RoboDK station: DensoAssemblyInverted.rdk

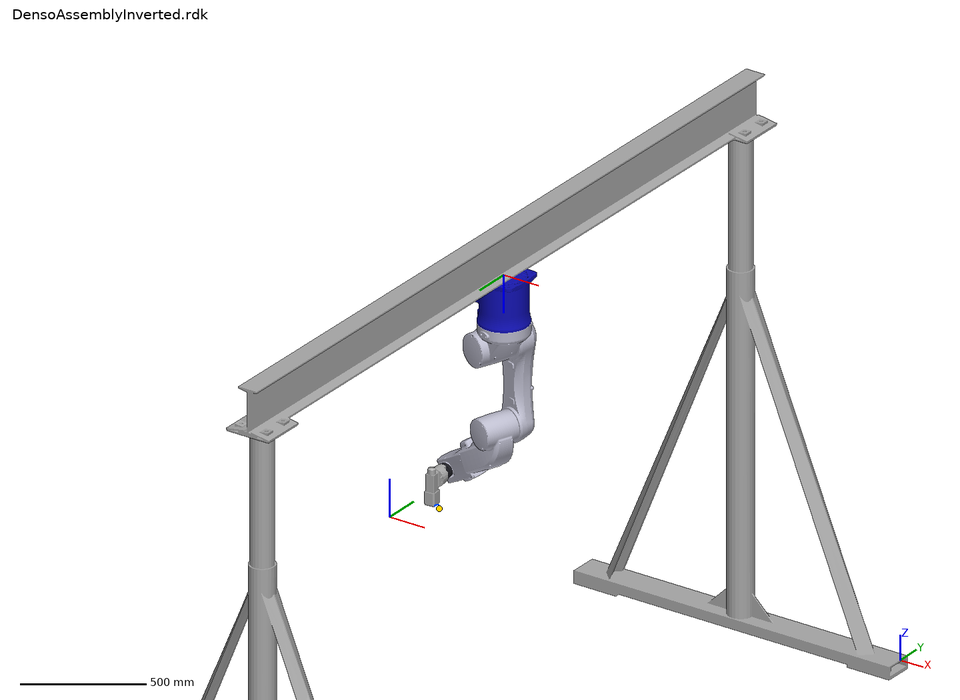
[picture v0: the station drawn from its stored meshes, robots at their saved joint values, targets as dots, program paths as lines]
Station DensoAssemblyInverted (saved by RoboDK 5.5.4). Poses are relative to the parent item; angles as X-Y-Z fixed-axis rotations.
Station parameters (name, value as stored): TAGS, ['Additive Manufacturing', 'Additive manufacturing'], LIN64
  - frame Denso VS-6577G-B Base at (0, 890, 2451.84) mm, rotated rx 180 ry 0 rz 0 deg
    - robot Denso VS-6577G-B: 6 axes, payload 7 kg, reach 854 mm, repeatability 0.03 mm, weight 36 kg
        modified DH rows (alpha deg, a mm, theta deg, d mm): 0, 0, 0, 335; -90, 75, -90, 0; 0, 365, -90, 0; -90, 90, 0, 405; 90, 0, 0, 0; -90, 0, 0, 80
        joint limits [-170, -100, -119, -190, -120, -360] to [170, 135, 169, 190, 120, 360]; home [0, 0, 90, 0, 0, 0]; saved at [-160.107, -3.776, 63.781, -103.06, 111.38, 57.53]
      - tool nozzle, TCP at (110, 10, 80) mm, rotated rx -90 ry 0 rz -90 deg, size 158.8 x 76.2 x 114.9 mm, geometry from nozzle.STEP
  - frame Reference at (-425.65, 710, 1340) mm
    - object Part at (-500, 0, 0) mm, size 120 x 120 x 160 mm, geometry from part.sld
  - machining project Print3D settings: /home/iRETI/RoboticsResearch/WallSection2.gcode | rotZ(0) | rotX(0)*rotY(0) | rotZ(0)
  - Python program Extruder (listed below)
  - Python program SimulateFinalResult (listed below)
  - object Gantry Assembly at (-570, 330, -20) mm, rotated rx 90 ry 0 rz 0 deg, size 1524 x 2402.4 x 3505.2 mm, geometry from Gantry Assembly.STEP
  - program Print3D (214 instructions, listed below)
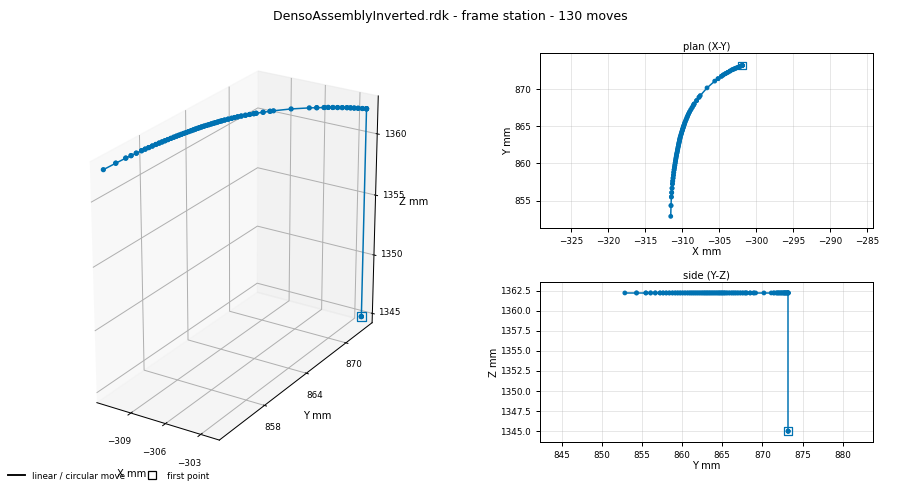
[picture p0: tool path of DensoAssemblyInverted.rdk in frame station, 130 of 130 moves have a stored position in this frame; points joined in program order, loops and branches not executed]

--- Python program Extruder ---
# This macro allows simulating a 3D printing extruder
# The macro will output spray gun statistics
#
# More information about the RoboDK API here:
# https://robodk.com/doc/en/RoboDK-API.html
# For more information visit:
# http://www.robodk.com/doc/en/PythonAPI/robolink.html
#
# Define the default action (0 to deactivate, +1 to activate, -1 to clear any spray gun simulation)
# Setting it to None will display a message
ACTION = None
# Check if we are running this program inside another program and passing arguments
import sys
if len(sys.argv) > 1:
    ACTION = float(sys.argv[1])
    # For faster speed: igone values greater than 0
    if ACTION > 0:
        quit()

from robolink import *    # API to communicate with RoboDK
from robodk import *      # basic matrix operations
RDK = Robolink()

# quit if we are not in simulation mode
if RDK.RunMode() != RUNMODE_SIMULATE:
    quit()

# Get any previously added spray gun simulations and display statistics (spray on the part vs spray falling out of the part)
existing_material_simulation = False
info, stats_data = RDK.Spray_GetStats()
if stats_data.size(1) > 0:
    print("Spray gun statistics:")
    print(info)
    print(stats_data.tr())
    existing_material_simulation = True
    # # Diplay statistics
    # RDK.ShowMessage("Material used: %.1f%%<br>Material waisted: %.1f%%<br>Total particles: %.1f" % (data[1,0],data[2,0],data[3,0]), True)
    # # Clear previous spray
    # RDK.Spray_Clear()

# If the default ACTION is None, display a message to activate/deactivate the spray gun
if ACTION is None:
    print('Note: This macro can be called as Extruder(0) to turn it ON or Extruder(-1) to turn it OFF')
    entry = mbox('Turn Extruder ON or OFF', ('On', '0'), ('Off', '-1'))
    if not entry:
        quit()
    ACTION = int(entry)

if ACTION < 0:
    # Turn material deposition off
    # Select Escape to delete existing material simulations
    #RDK.Spray_Clear()
    RDK.Spray_SetState(SPRAY_OFF)

elif ACTION >= 0:

    if existing_material_simulation:
        # Select Esc key to delete existing material simulations and force a new type of spray gun simulation
        RDK.Spray_SetState(SPRAY_ON)
        exit()


    # Create a new spray gun object in RoboDK for material deposition (3D printing simulation)
    # by using RDK.Spray_Add(tool, object, options_command, volume, geometry)
    # tool: tool item (TCP) to use
    # object: object to project the particles
    # options_command (optional): string to specify options. Example:
    #     STEP=AxB: Defines the grid to be projected 1x1 means only one line of particle projection (for example, for welding)
    #     PARTICLE: Defines the shape and size of particle (sphere or particle), unless a specific geometry is provided:
    #       a- SPHERE(radius, facets)
    #       b- SPHERE(radius, facets, scalex, scaley, scalez)
    #       b- CUBE(sizex, sizey, sizez)
    #     RAND=factor: Defines a random factor factor 0 means that the particles are not deposited randomly
    #     ELLYPSE: defines the volume as an ellypse (default)
    #     RECTANGLE: defines the volume as a rectangle
    #     PROJECT: project the particles to the surface (default) (for welding, painting or scanning)
    #     NO_PROJECT: does not project the particles to the surface (for example, for 3D printing)
    #
    # volume (optional): Matrix of parameters defining the volume of the spray gun
    # geometry (optional): Matrix of vertices defining the triangles.


    diameter = 22.225 # in mm
    detail = 8 # number of rings of detail to display the sphere
    scale = '1,1,0.5' # scale the particle in 0.5 along the tool Z axis (simulating gravity effect)
    options_command = "ELLYPSE NO_PROJECT PARTICLE=SPHERE(%.3f,%.0f,%s)" % (diameter, detail, scale) # simulate
    #options_command = "PARTICLE=CUBE(10,10,2) STEP=8x8"
    #options_command = "PARTICLE=SPHERE(4,8) STEP=8x8"
    #options_command = "PARTICLE=SPHERE(4,8,1,1,0.1) STEP=8x8 RAND=3"

    # Example commands for welding:
    # options_command = "PROJECT PARTICLE=SPHERE(4,8)"
    # options_command = PARTICLE=SPHERE(4,8) STEP=1x0

    tool = 0    # auto detect active tool
    obj = 0     # auto detect object in active reference frame

    # Material is deposited at 0,0,0 with respect to the TCP coordinates
    close_param = [0,0,0,  0,0,0,  0,0,0,     0.7,0.5,0.8,1] # color as RGBA
    far_param   = [0,0,0,  0,0,0,  0,0,0,     0.7,0.5,0.8,1] # color as RGBA
    volume = Mat([close_param, far_param])
    RDK.Spray_Add(tool, obj, options_command, volume.tr())
    RDK.Spray_SetState(SPRAY_ON)

--- Python program SimulateFinalResult ---
# This script will simulate the final result of the 3D printed part using the Spray function

# Or visit: http://www.robodk.com/doc/PythonAPI/
# Note: you do not need to keep a copy of this file, your python script is saved with the station
from robolink import *    # API to communicate with RoboDK
from robodk import *      # basic matrix operations


RENDER = True      # Set to False
STEP_MM = 2         # Detail step in MM for linear moves
STEP_DEG = 2        # Detail step in DEG for joint moves

# Start a connection with the RoboDK API
RDK = Robolink()

# Select the first/only robot in the cell:
program = RDK.ItemUserPick('Select a program to simulate', ITEM_TYPE_PROGRAM)
if not program.Valid():
    raise Exception("No program available")

# Get the robot
robot = RDK.Item('', ITEM_TYPE_ROBOT)
#robot = program.getLink(ITEM_TYPE_ROBOT) # available in newer versions
if not robot.Valid():
    raise Exception("No robot available")

progname = program.Name()
print("Using program %s" % progname)


# Get the program as a list of joint values
tool = robot.getLink(ITEM_TYPE_TOOL)
progok_jlist = program.InstructionListJoints(STEP_MM, STEP_DEG)
progok = progok_jlist[0] # progok: String that indicates if there are any issues with the program
jlist = progok_jlist[1]  # jlist: list of joints

# Check that the program is correct and has at least a movement
njoints = jlist.size(1)
if njoints < 1:
    raise Exception("Program %s has no movements" % name)

# Check if there are any issues with the program:
if progok != "Success":
    raise Exception("Problems with program %s: %s." %(name, progok))

# Reset any material deposition simulation
RDK.Spray_Clear()

robot.setPoseTool(tool)

# Start material deposition simulation according to the Extruder script
RDK.RunProgram('Extruder(0)')
# Alternatively:
#RDK.Item('Extruder', ITEM_TYPE_PYTHON).RunProgram([1])

if not RENDER:
    RDK.Render(False)

# Iterate through all joints in the matrix and check for collisions
njoints_all = jlist.size(1)
for i in range(njoints_all):
    ji = jlist[:,i].tolist()

    # Update the robot to a new position (it will create a new particle)
    robot.setJoints(ji)
    if not RENDER:
        # If Render is turned off (faster) update the position to draw a new particle
        RDK.Update()

    # Show a message in the RoboDK status bar from time to time
    if i % 10 == 0:
        msg = "Quick material deposition simulation for %s (%.1f %%)" % (progname, 100.0*(i/njoints_all))
        print(msg)
        RDK.ShowMessage(msg, False)

    # Render from time to time even if we have render deactivated
    if not RENDER and i % 500 == 0:
        RDK.Render()

RDK.Render(True)
msg = "Done"
print("Done")
RDK.ShowMessage(msg, False)

--- program Print3D (robot Denso VS-6577G-B) ---
  Call M_RunCode(107)
  Call M_RunCode(104)
  Set speed (83.3 mm/s)
  Set speed (1000.0 mm/s)
  Set Ref.: Reference
  Set Tool: nozzle
  Show nozzle
  MoveJ 1 to (123.76, 163.21, 5) mm, rotated rx -180 ry 0 rz -175 deg; joints [-156.49, -1.48, 58.301, -106.555, 113.546, 53.347]
  MoveL 2 to (123.76, 163.21, 5) mm, rotated rx -180 ry 0 rz -175 deg; joints [-156.49, -1.48, 58.301, -106.555, 113.546, 53.347]
  Call Extruder(-1)
  MoveL 3 to (123.76, 163.21, 5) mm, rotated rx -180 ry 0 rz -175 deg; joints [-156.49, -1.48, 58.301, -106.555, 113.546, 53.347]
  Call M_RunCode(109)
  Call M_RunCode(82)
  Call Extruder(0.00000)
  Set speed (130.0 mm/s)
  MoveL 4 to (123.76, 163.21, 22.22) mm, rotated rx 180 ry 0 rz -175 deg; joints [-156.49, -3.989, 63.978, -105.199, 114.413, 56.682]
  Call Extruder(-2.00000)
  Set speed (40.0 mm/s)
  MoveL 5 to (123.76, 163.21, 22.22) mm, rotated rx 180 ry 0 rz -175 deg; joints [-156.49, -3.989, 63.978, -105.199, 114.413, 56.682]
  Call Extruder(0.00000)
  Set speed (130.0 mm/s)
  MoveL 6 to (123.76, 163.21, 22.22) mm, rotated rx 180 ry 0 rz -175 deg; joints [-156.49, -3.989, 63.978, -105.199, 114.413, 56.682]
  Call Extruder(2.00000)
  Set speed (40.0 mm/s)
  MoveL 7 to (123.76, 163.21, 22.22) mm, rotated rx 180 ry 0 rz -175 deg; joints [-156.49, -3.989, 63.978, -105.199, 114.413, 56.682]
  Set speed (30.0 mm/s)
  MoveL 8 to (123.76, 163.21, 22.22) mm, rotated rx 180 ry 0 rz -175 deg; joints [-156.49, -3.989, 63.978, -105.199, 114.413, 56.682]
  Call Extruder(2.38024)
  MoveL 9 to (123.47, 163.09, 22.22) mm, rotated rx -180 ry 0 rz -175 deg; joints [-156.527, -3.957, 63.948, -105.176, 114.383, 56.694]
  MoveL 10 to (123.47, 163.09, 22.22) mm, rotated rx -180 ry 0 rz -175 deg; joints [-156.527, -3.957, 63.948, -105.176, 114.383, 56.694]
  Call Extruder(2.76227)
  MoveL 11 to (123.18, 162.97, 22.22) mm, rotated rx -180 ry 0 rz -175 deg; joints [-156.564, -3.924, 63.918, -105.153, 114.353, 56.706]
  MoveL 12 to (123.18, 162.97, 22.22) mm, rotated rx -180 ry 0 rz -175 deg; joints [-156.564, -3.924, 63.918, -105.153, 114.353, 56.706]
  Call Extruder(3.11872)
  MoveL 13 to (122.91, 162.85, 22.23) mm, rotated rx -180 ry 0 rz -175 deg; joints [-156.598, -3.894, 63.891, -105.131, 114.325, 56.717]
  MoveL 14 to (122.91, 162.85, 22.23) mm, rotated rx -180 ry 0 rz -175 deg; joints [-156.598, -3.894, 63.891, -105.131, 114.325, 56.717]
  Call Extruder(3.44932)
  MoveL 15 to (122.66, 162.74, 22.23) mm, rotated rx -180 ry 0 rz -175 deg; joints [-156.629, -3.867, 63.865, -105.111, 114.299, 56.727]
  MoveL 16 to (122.66, 162.74, 22.23) mm, rotated rx -180 ry 0 rz -175 deg; joints [-156.629, -3.867, 63.865, -105.111, 114.299, 56.727]
  Call Extruder(3.78134)
  MoveL 17 to (122.41, 162.64, 22.23) mm, rotated rx 180 ry 0 rz -175 deg; joints [-156.661, -3.839, 63.84, -105.091, 114.273, 56.737]
  MoveL 18 to (122.41, 162.64, 22.23) mm, rotated rx 180 ry 0 rz -175 deg; joints [-156.661, -3.839, 63.84, -105.091, 114.273, 56.737]
  Call Extruder(4.21321)
  MoveL 19 to (122.11, 162.46, 22.22) mm, rotated rx -180 ry 0 rz -175 deg; joints [-156.706, -3.808, 63.811, -105.063, 114.236, 56.751]
  MoveL 20 to (122.11, 162.46, 22.22) mm, rotated rx -180 ry 0 rz -175 deg; joints [-156.706, -3.808, 63.811, -105.063, 114.236, 56.751]
  Call Extruder(4.64692)
  MoveL 21 to (121.8, 162.29, 22.22) mm, rotated rx -180 ry 0 rz -175 deg; joints [-156.752, -3.777, 63.782, -105.035, 114.199, 56.765]
  MoveL 22 to (121.8, 162.29, 22.22) mm, rotated rx -180 ry 0 rz -175 deg; joints [-156.752, -3.777, 63.782, -105.035, 114.199, 56.765]
  Call Extruder(5.08247)
  MoveL 23 to (121.5, 162.11, 22.22) mm, rotated rx -180 ry 0 rz -175 deg; joints [-156.797, -3.746, 63.754, -105.006, 114.162, 56.778]
  MoveL 24 to (121.5, 162.11, 22.22) mm, rotated rx -180 ry 0 rz -175 deg; joints [-156.797, -3.746, 63.754, -105.006, 114.162, 56.778]
  Call Extruder(5.51986)
  MoveL 25 to (121.19, 161.94, 22.22) mm, rotated rx -180 ry 0 rz -175 deg; joints [-156.842, -3.715, 63.725, -104.978, 114.125, 56.792]
  MoveL 26 to (121.19, 161.94, 22.22) mm, rotated rx -180 ry 0 rz -175 deg; joints [-156.842, -3.715, 63.725, -104.978, 114.125, 56.792]
  Call Extruder(5.89660)
  MoveL 27 to (120.95, 161.76, 22.23) mm, rotated rx -180 ry 0 rz -175 deg; joints [-156.883, -3.691, 63.704, -104.953, 114.091, 56.804]
  MoveL 28 to (120.95, 161.76, 22.23) mm, rotated rx -180 ry 0 rz -175 deg; joints [-156.883, -3.691, 63.704, -104.953, 114.091, 56.804]
  Call Extruder(6.59657)
  MoveL 29 to (120.5, 161.43, 22.22) mm, rotated rx 180 ry 0 rz -175 deg; joints [-156.96, -3.649, 63.664, -104.905, 114.027, 56.826]
  MoveL 30 to (120.5, 161.43, 22.22) mm, rotated rx 180 ry 0 rz -175 deg; joints [-156.96, -3.649, 63.664, -104.905, 114.027, 56.826]
  Call Extruder(7.29934)
  MoveL 31 to (120.05, 161.1, 22.22) mm, rotated rx 180 ry 0 rz -175 deg; joints [-157.037, -3.606, 63.625, -104.858, 113.964, 56.848]
  Call Extruder(9.03811)
  MoveL 32 to (119.01, 160.19, 22.22) mm, rotated rx -180 ry 0 rz -175 deg; joints [-157.235, -3.517, 63.542, -104.736, 113.799, 56.904]
  Call Extruder(10.77694)
  MoveL 33 to (118.1, 159.15, 22.22) mm, rotated rx 180 ry 0 rz -175 deg; joints [-157.444, -3.451, 63.481, -104.61, 113.625, 56.959]
  Call Extruder(11.12832)
  MoveL 34 to (117.93, 158.93, 22.22) mm, rotated rx -180 ry 0 rz -175 deg; joints [-157.488, -3.441, 63.472, -104.584, 113.589, 56.97]
  MoveL 35 to (117.93, 158.93, 22.22) mm, rotated rx -180 ry 0 rz -175 deg; joints [-157.488, -3.441, 63.472, -104.584, 113.589, 56.97]
  Call Extruder(11.82828)
  MoveL 36 to (117.61, 158.48, 22.22) mm, rotated rx -180 ry 0 rz -175 deg; joints [-157.574, -3.422, 63.454, -104.532, 113.517, 56.992]
  MoveL 37 to (117.61, 158.48, 22.22) mm, rotated rx -180 ry 0 rz -175 deg; joints [-157.574, -3.422, 63.454, -104.532, 113.517, 56.992]
  Call Extruder(12.52544)
  MoveL 38 to (117.28, 158.03, 22.22) mm, rotated rx -180 ry 0 rz -175 deg; joints [-157.661, -3.402, 63.435, -104.48, 113.445, 57.014]
  MoveL 39 to (117.28, 158.03, 22.22) mm, rotated rx -180 ry 0 rz -175 deg; joints [-157.661, -3.402, 63.435, -104.48, 113.445, 57.014]
  Call Extruder(12.77229)
  MoveL 40 to (117.18, 157.85, 22.22) mm, rotated rx -180 ry 0 rz -175 deg; joints [-157.692, -3.398, 63.432, -104.461, 113.418, 57.021]
  MoveL 41 to (117.18, 157.85, 22.22) mm, rotated rx -180 ry 0 rz -175 deg; joints [-157.692, -3.398, 63.432, -104.461, 113.418, 57.021]
  Call Extruder(13.20785)
  MoveL 42 to (117, 157.55, 22.23) mm, rotated rx -180 ry 0 rz -175 deg; joints [-157.748, -3.391, 63.425, -104.428, 113.372, 57.035]
  MoveL 43 to (117, 157.55, 22.23) mm, rotated rx -180 ry 0 rz -175 deg; joints [-157.748, -3.391, 63.425, -104.428, 113.372, 57.035]
  Call Extruder(13.64157)
  MoveL 44 to (116.83, 157.25, 22.22) mm, rotated rx 180 ry 0 rz -175 deg; joints [-157.803, -3.384, 63.419, -104.395, 113.326, 57.049]
  MoveL 45 to (116.83, 157.25, 22.22) mm, rotated rx 180 ry 0 rz -175 deg; joints [-157.803, -3.384, 63.419, -104.395, 113.326, 57.049]
  Call Extruder(14.07344)
  MoveL 46 to (116.65, 156.94, 22.22) mm, rotated rx -180 ry 0 rz -175 deg; joints [-157.859, -3.377, 63.412, -104.362, 113.279, 57.062]
  MoveL 47 to (116.65, 156.94, 22.22) mm, rotated rx -180 ry 0 rz -175 deg; joints [-157.859, -3.377, 63.412, -104.362, 113.279, 57.062]
  Call Extruder(14.45383)
  MoveL 48 to (116.51, 156.66, 22.22) mm, rotated rx -180 ry 0 rz -175 deg; joints [-157.908, -3.373, 63.408, -104.332, 113.238, 57.074]
  MoveL 49 to (116.51, 156.66, 22.22) mm, rotated rx -180 ry 0 rz -175 deg; joints [-157.908, -3.373, 63.408, -104.332, 113.238, 57.074]
  Call Extruder(14.78446)
  MoveL 50 to (116.4, 156.42, 22.23) mm, rotated rx -180 ry 0 rz -175 deg; joints [-157.951, -3.372, 63.407, -104.307, 113.202, 57.084]
  MoveL 51 to (116.4, 156.42, 22.23) mm, rotated rx -180 ry 0 rz -175 deg; joints [-157.951, -3.372, 63.407, -104.307, 113.202, 57.084]
  Call Extruder(15.11366)
  MoveL 52 to (116.3, 156.17, 22.23) mm, rotated rx -180 ry 0 rz -175 deg; joints [-157.994, -3.371, 63.407, -104.281, 113.165, 57.094]
  MoveL 53 to (116.3, 156.17, 22.23) mm, rotated rx -180 ry 0 rz -175 deg; joints [-157.994, -3.371, 63.407, -104.281, 113.165, 57.094]
  Call Extruder(15.49565)
  MoveL 54 to (116.17, 155.88, 22.22) mm, rotated rx 180 ry 0 rz -175 deg; joints [-158.045, -3.371, 63.406, -104.252, 113.123, 57.106]
  MoveL 55 to (116.17, 155.88, 22.22) mm, rotated rx 180 ry 0 rz -175 deg; joints [-158.045, -3.371, 63.406, -104.252, 113.123, 57.106]
  Call Extruder(15.87585)
  MoveL 56 to (116.05, 155.58, 22.22) mm, rotated rx 180 ry 0 rz -175 deg; joints [-158.095, -3.37, 63.406, -104.222, 113.081, 57.118]
  MoveL 57 to (116.05, 155.58, 22.22) mm, rotated rx 180 ry 0 rz -175 deg; joints [-158.095, -3.37, 63.406, -104.222, 113.081, 57.118]
  Call Extruder(16.18353)
  MoveL 58 to (115.96, 155.34, 22.22) mm, rotated rx -180 ry 0 rz -175 deg; joints [-158.136, -3.371, 63.407, -104.198, 113.046, 57.127]
  MoveL 59 to (115.96, 155.34, 22.22) mm, rotated rx -180 ry 0 rz -175 deg; joints [-158.136, -3.371, 63.407, -104.198, 113.046, 57.127]
  Call Extruder(16.41988)
  MoveL 60 to (115.9, 155.15, 22.22) mm, rotated rx 180 ry 0 rz -175 deg; joints [-158.168, -3.373, 63.408, -104.179, 113.02, 57.134]
  MoveL 61 to (115.9, 155.15, 22.22) mm, rotated rx 180 ry 0 rz -175 deg; joints [-158.168, -3.373, 63.408, -104.179, 113.02, 57.134]
  Call Extruder(16.65518)
  MoveL 62 to (115.84, 154.97, 22.22) mm, rotated rx -180 ry 0 rz -175 deg; joints [-158.199, -3.375, 63.41, -104.161, 112.993, 57.141]
  MoveL 63 to (115.84, 154.97, 22.22) mm, rotated rx -180 ry 0 rz -175 deg; joints [-158.199, -3.375, 63.41, -104.161, 112.993, 57.141]
  Call Extruder(16.88943)
  MoveL 64 to (115.78, 154.78, 22.22) mm, rotated rx 180 ry 0 rz -175 deg; joints [-158.231, -3.377, 63.412, -104.142, 112.967, 57.148]
  MoveL 65 to (115.78, 154.78, 22.22) mm, rotated rx 180 ry 0 rz -175 deg; joints [-158.231, -3.377, 63.412, -104.142, 112.967, 57.148]
  Call Extruder(17.12262)
  MoveL 66 to (115.72, 154.59, 22.22) mm, rotated rx 180 ry 0 rz -175 deg; joints [-158.262, -3.379, 63.414, -104.124, 112.94, 57.155]
  MoveL 67 to (115.72, 154.59, 22.22) mm, rotated rx 180 ry 0 rz -175 deg; joints [-158.262, -3.379, 63.414, -104.124, 112.94, 57.155]
  Call Extruder(17.37548)
  MoveL 68 to (115.65, 154.38, 22.22) mm, rotated rx -180 ry 0 rz -175 deg; joints [-158.296, -3.381, 63.416, -104.103, 112.911, 57.163]
  MoveL 69 to (115.65, 154.38, 22.22) mm, rotated rx -180 ry 0 rz -175 deg; joints [-158.296, -3.381, 63.416, -104.103, 112.911, 57.163]
  Call Extruder(17.64775)
  MoveL 70 to (115.58, 154.16, 22.23) mm, rotated rx -180 ry 0 rz -175 deg; joints [-158.334, -3.384, 63.419, -104.082, 112.88, 57.171]
  MoveL 71 to (115.58, 154.16, 22.23) mm, rotated rx -180 ry 0 rz -175 deg; joints [-158.334, -3.384, 63.419, -104.082, 112.88, 57.171]
  Call Extruder(17.91868)
  MoveL 72 to (115.52, 153.94, 22.23) mm, rotated rx -180 ry 0 rz -175 deg; joints [-158.371, -3.387, 63.422, -104.06, 112.849, 57.18]
  MoveL 73 to (115.52, 153.94, 22.23) mm, rotated rx -180 ry 0 rz -175 deg; joints [-158.371, -3.387, 63.422, -104.06, 112.849, 57.18]
  Call Extruder(18.18828)
  MoveL 74 to (115.45, 153.71, 22.22) mm, rotated rx -180 ry 0 rz -175 deg; joints [-158.408, -3.39, 63.424, -104.038, 112.818, 57.188]
  MoveL 75 to (115.45, 153.71, 22.22) mm, rotated rx -180 ry 0 rz -175 deg; joints [-158.408, -3.39, 63.424, -104.038, 112.818, 57.188]
  Call Extruder(18.45654)
  MoveL 76 to (115.38, 153.49, 22.22) mm, rotated rx -180 ry 0 rz -175 deg; joints [-158.445, -3.393, 63.427, -104.016, 112.786, 57.196]
  MoveL 77 to (115.38, 153.49, 22.22) mm, rotated rx -180 ry 0 rz -175 deg; joints [-158.445, -3.393, 63.427, -104.016, 112.786, 57.196]
  Call Extruder(18.69554)
  MoveL 78 to (115.34, 153.28, 22.22) mm, rotated rx -180 ry 0 rz -175 deg; joints [-158.478, -3.398, 63.432, -103.997, 112.759, 57.203]
  MoveL 79 to (115.34, 153.28, 22.22) mm, rotated rx -180 ry 0 rz -175 deg; joints [-158.478, -3.398, 63.432, -103.997, 112.759, 57.203]
  Call Extruder(18.93348)
  MoveL 80 to (115.29, 153.08, 22.22) mm, rotated rx 180 ry 0 rz -175 deg; joints [-158.511, -3.403, 63.436, -103.978, 112.731, 57.21]
  MoveL 81 to (115.29, 153.08, 22.22) mm, rotated rx 180 ry 0 rz -175 deg; joints [-158.511, -3.403, 63.436, -103.978, 112.731, 57.21]
  Call Extruder(19.17035)
  MoveL 82 to (115.25, 152.88, 22.22) mm, rotated rx -180 ry 0 rz -175 deg; joints [-158.544, -3.408, 63.441, -103.959, 112.703, 57.217]
  MoveL 83 to (115.25, 152.88, 22.22) mm, rotated rx -180 ry 0 rz -175 deg; joints [-158.544, -3.408, 63.441, -103.959, 112.703, 57.217]
  Call Extruder(19.40615)
  MoveL 84 to (115.2, 152.67, 22.23) mm, rotated rx -180 ry 0 rz -175 deg; joints [-158.577, -3.413, 63.445, -103.94, 112.675, 57.225]
  MoveL 85 to (115.2, 152.67, 22.23) mm, rotated rx -180 ry 0 rz -175 deg; joints [-158.577, -3.413, 63.445, -103.94, 112.675, 57.225]
  Call Extruder(19.66605)
  MoveL 86 to (115.16, 152.45, 22.22) mm, rotated rx -180 ry 0 rz -175 deg; joints [-158.613, -3.418, 63.451, -103.919, 112.645, 57.232]
  MoveL 87 to (115.16, 152.45, 22.22) mm, rotated rx -180 ry 0 rz -175 deg; joints [-158.613, -3.418, 63.451, -103.919, 112.645, 57.232]
  Call Extruder(19.94972)
  MoveL 88 to (115.11, 152.2, 22.22) mm, rotated rx -180 ry 0 rz -175 deg; joints [-158.653, -3.425, 63.457, -103.895, 112.611, 57.241]
  MoveL 89 to (115.11, 152.2, 22.22) mm, rotated rx -180 ry 0 rz -175 deg; joints [-158.653, -3.425, 63.457, -103.895, 112.611, 57.241]
  Call Extruder(20.23193)
  MoveL 90 to (115.06, 151.95, 22.22) mm, rotated rx -180 ry 0 rz -175 deg; joints [-158.693, -3.432, 63.463, -103.872, 112.577, 57.249]
  MoveL 91 to (115.06, 151.95, 22.22) mm, rotated rx -180 ry 0 rz -175 deg; joints [-158.693, -3.432, 63.463, -103.872, 112.577, 57.249]
  Call Extruder(20.51271)
  MoveL 92 to (115.01, 151.7, 22.23) mm, rotated rx -180 ry 0 rz -175 deg; joints [-158.733, -3.438, 63.469, -103.849, 112.544, 57.258]
  MoveL 93 to (115.01, 151.7, 22.23) mm, rotated rx -180 ry 0 rz -175 deg; joints [-158.733, -3.438, 63.469, -103.849, 112.544, 57.258]
  Call Extruder(20.79205)
  MoveL 94 to (114.96, 151.45, 22.23) mm, rotated rx -180 ry 0 rz -175 deg; joints [-158.773, -3.445, 63.475, -103.826, 112.51, 57.266]
  MoveL 95 to (114.96, 151.45, 22.23) mm, rotated rx -180 ry 0 rz -175 deg; joints [-158.773, -3.445, 63.475, -103.826, 112.51, 57.266]
  Call Extruder(21.06994)
  MoveL 96 to (114.91, 151.2, 22.22) mm, rotated rx -180 ry 0 rz -175 deg; joints [-158.813, -3.451, 63.481, -103.803, 112.476, 57.275]
  MoveL 97 to (114.91, 151.2, 22.22) mm, rotated rx -180 ry 0 rz -175 deg; joints [-158.813, -3.451, 63.481, -103.803, 112.476, 57.275]
  Call Extruder(21.34639)
  MoveL 98 to (114.86, 150.95, 22.22) mm, rotated rx -180 ry 0 rz -175 deg; joints [-158.852, -3.458, 63.488, -103.779, 112.443, 57.283]
  MoveL 99 to (114.86, 150.95, 22.22) mm, rotated rx -180 ry 0 rz -175 deg; joints [-158.852, -3.458, 63.488, -103.779, 112.443, 57.283]
  Call Extruder(21.65140)
  MoveL 100 to (114.81, 150.67, 22.23) mm, rotated rx -180 ry 0 rz -175 deg; joints [-158.897, -3.466, 63.495, -103.754, 112.405, 57.292]
  MoveL 101 to (114.81, 150.67, 22.23) mm, rotated rx -180 ry 0 rz -175 deg; joints [-158.897, -3.466, 63.495, -103.754, 112.405, 57.292]
  Call Extruder(21.98479)
  MoveL 102 to (114.76, 150.37, 22.22) mm, rotated rx -180 ry 0 rz -175 deg; joints [-158.945, -3.476, 63.504, -103.726, 112.364, 57.302]
  MoveL 103 to (114.76, 150.37, 22.22) mm, rotated rx -180 ry 0 rz -175 deg; joints [-158.945, -3.476, 63.504, -103.726, 112.364, 57.302]
  Call Extruder(22.31647)
  MoveL 104 to (114.71, 150.06, 22.22) mm, rotated rx -180 ry 0 rz -175 deg; joints [-158.993, -3.485, 63.513, -103.698, 112.324, 57.312]
  MoveL 105 to (114.71, 150.06, 22.22) mm, rotated rx -180 ry 0 rz -175 deg; joints [-158.993, -3.485, 63.513, -103.698, 112.324, 57.312]
  Call Extruder(22.64643)
  MoveL 106 to (114.66, 149.76, 22.22) mm, rotated rx -180 ry 0 rz -175 deg; joints [-159.042, -3.495, 63.522, -103.67, 112.283, 57.322]
  MoveL 107 to (114.66, 149.76, 22.22) mm, rotated rx -180 ry 0 rz -175 deg; joints [-159.042, -3.495, 63.522, -103.67, 112.283, 57.322]
  Call Extruder(22.97467)
  MoveL 108 to (114.62, 149.45, 22.22) mm, rotated rx -180 ry 0 rz -175 deg; joints [-159.09, -3.504, 63.531, -103.642, 112.242, 57.332]
  MoveL 109 to (114.62, 149.45, 22.22) mm, rotated rx -180 ry 0 rz -175 deg; joints [-159.09, -3.504, 63.531, -103.642, 112.242, 57.332]
  Call Extruder(23.30119)
  MoveL 110 to (114.57, 149.14, 22.22) mm, rotated rx 180 ry 0 rz -175 deg; joints [-159.138, -3.514, 63.539, -103.614, 112.201, 57.342]
  MoveL 111 to (114.57, 149.14, 22.22) mm, rotated rx 180 ry 0 rz -175 deg; joints [-159.138, -3.514, 63.539, -103.614, 112.201, 57.342]
  Call Extruder(23.66827)
  MoveL 112 to (114.52, 148.8, 22.22) mm, rotated rx -180 ry 0 rz -175 deg; joints [-159.193, -3.526, 63.55, -103.583, 112.155, 57.353]
  MoveL 113 to (114.52, 148.8, 22.22) mm, rotated rx -180 ry 0 rz -175 deg; joints [-159.193, -3.526, 63.55, -103.583, 112.155, 57.353]
  Call Extruder(24.07571)
  MoveL 114 to (114.47, 148.41, 22.22) mm, rotated rx -180 ry 0 rz -175 deg; joints [-159.253, -3.54, 63.563, -103.548, 112.104, 57.366]
  MoveL 115 to (114.47, 148.41, 22.22) mm, rotated rx -180 ry 0 rz -175 deg; joints [-159.253, -3.54, 63.563, -103.548, 112.104, 57.366]
  Call Extruder(24.48110)
  MoveL 116 to (114.43, 148.02, 22.23) mm, rotated rx 180 ry 0 rz -175 deg; joints [-159.314, -3.554, 63.576, -103.513, 112.052, 57.378]
  MoveL 117 to (114.43, 148.02, 22.23) mm, rotated rx 180 ry 0 rz -175 deg; joints [-159.314, -3.554, 63.576, -103.513, 112.052, 57.378]
  Call Extruder(24.88445)
  MoveL 118 to (114.38, 147.63, 22.22) mm, rotated rx -180 ry 0 rz -175 deg; joints [-159.375, -3.568, 63.589, -103.478, 112.001, 57.39]
  MoveL 119 to (114.38, 147.63, 22.22) mm, rotated rx -180 ry 0 rz -175 deg; joints [-159.375, -3.568, 63.589, -103.478, 112.001, 57.39]
  Call Extruder(25.28574)
  MoveL 120 to (114.34, 147.25, 22.23) mm, rotated rx -180 ry 0 rz -175 deg; joints [-159.435, -3.582, 63.602, -103.443, 111.95, 57.402]
  MoveL 121 to (114.34, 147.25, 22.23) mm, rotated rx -180 ry 0 rz -175 deg; joints [-159.435, -3.582, 63.602, -103.443, 111.95, 57.402]
  Call Extruder(25.89062)
  MoveL 122 to (114.29, 146.66, 22.22) mm, rotated rx -180 ry 0 rz -175 deg; joints [-159.526, -3.606, 63.625, -103.391, 111.873, 57.42]
  MoveL 123 to (114.29, 146.66, 22.22) mm, rotated rx -180 ry 0 rz -175 deg; joints [-159.526, -3.606, 63.625, -103.391, 111.873, 57.42]
  Call Extruder(26.49235)
  MoveL 124 to (114.24, 146.07, 22.22) mm, rotated rx 180 ry 0 rz -175 deg; joints [-159.617, -3.63, 63.647, -103.339, 111.796, 57.437]
  MoveL 125 to (114.24, 146.07, 22.22) mm, rotated rx 180 ry 0 rz -175 deg; joints [-159.617, -3.63, 63.647, -103.339, 111.796, 57.437]
  Call Extruder(27.09093)
  MoveL 126 to (114.2, 145.48, 22.22) mm, rotated rx -180 ry 0 rz -175 deg; joints [-159.708, -3.654, 63.669, -103.287, 111.718, 57.455]
  MoveL 127 to (114.2, 145.48, 22.22) mm, rotated rx -180 ry 0 rz -175 deg; joints [-159.708, -3.654, 63.669, -103.287, 111.718, 57.455]
  Call Extruder(28.26271)
  MoveL 128 to (114.15, 144.32, 22.23) mm, rotated rx -180 ry 0 rz -175 deg; joints [-159.886, -3.707, 63.718, -103.186, 111.568, 57.489]
  MoveL 129 to (114.15, 144.32, 22.23) mm, rotated rx -180 ry 0 rz -175 deg; joints [-159.886, -3.707, 63.718, -103.186, 111.568, 57.489]
  Call Extruder(29.72057)
  MoveL 130 to (114.11, 142.86, 22.22) mm, rotated rx -180 ry 0 rz -175 deg; joints [-160.107, -3.776, 63.781, -103.06, 111.38, 57.53]
  Call Extruder(115.61408)
  Call Extruder(116.48916)
